(* PLC project testproj, Beckhoff Automation GmbH TwinCAT PLC Control 3.5.20.50 *)
(* stored: creationDateTime 2025-07-01T11:02:16.1300929, modificationDateTime 2025-07-01T11:02:16.1300929 *)

FUNCTION_BLOCK AnaMon
  VAR_INPUT
    WQC : BYTE;
    OSLevel : BYTE;
    V : REAL;
    VSclMin : REAL;
    VSclMax : REAL;
    VUnit : INT;
    VAHEn : BOOL;
    VWHEn : BOOL;
    VTHEn : BOOL;
    VTLEn : BOOL;
    VWLEn : BOOL;
    VALEn : BOOL;
  END_VAR
  VAR_OUTPUT
    VAHAct : BOOL;
    VWHAct : BOOL;
    VTHAct : BOOL;
    VTLAct : BOOL;
    VWLAct : BOOL;
    VALAct : BOOL;
  END_VAR
  VAR
    VAHLim : REAL;
    VWHLim : REAL;
    VTHLim : REAL;
    VTLLim : REAL;
    VWLLim : REAL;
    VALLim : REAL;
  END_VAR

            
// Copy MTP base variables to local temporaries (READ access)


VAHAct := vOut >= alarmHigh;
VWHAct := vOut >= warningHigh;
VTHAct := vOut >= toleranceHigh;
VTLAct := vOut <= toleranceLow;
VWLAct := vOut <= warningLow;
VALAct := vOut <= alarmLow;

// Copy local temporaries back to MTP base variables (WRITE access)

        
END_FUNCTION_BLOCK

FUNCTION_BLOCK BinMon
  VAR_INPUT
    wQC : BYTE;
    vState0 : STRING;
    vState1 : STRING;
    oSLevel : BYTE;
    vFlutEn : BOOL;
  END_VAR
  VAR_OUTPUT
    vFlutAct : BOOL;
  END_VAR
  VAR
    vFlutCnt : INT;
  END_VAR

            
// Copy MTP base variables to local temporaries (READ access)



// Copy local temporaries back to MTP base variables (WRITE access)

        
END_FUNCTION_BLOCK

FUNCTION_BLOCK LockView4
  VAR_INPUT
    wQC : BYTE;
    logic : BOOL;
    in1En : BOOL;
    in1 : BOOL;
    in1QC : BYTE;
    in1Inv : BOOL;
    in1Txt : STRING;
    in2En : BOOL;
    in2 : BOOL;
    in2QC : BYTE;
    in2Inv : BOOL;
    in2Txt : STRING;
    in3En : BOOL;
    in3 : BOOL;
    in3QC : BYTE;
    in3Inv : BOOL;
    in3Txt : STRING;
    in4En : BOOL;
    in4 : BOOL;
    in4QC : BYTE;
    in4Inv : BOOL;
    in4Txt : STRING;
  END_VAR
  VAR_OUTPUT
    out : BOOL;
    outQC : STRING;
  END_VAR

            
// Copy MTP base variables to local temporaries (READ access)



// Copy local temporaries back to MTP base variables (WRITE access)

        
END_FUNCTION_BLOCK

FUNCTION_BLOCK MonAnaDrv

            
// Copy MTP base variables to local temporaries (READ access)



// Copy local temporaries back to MTP base variables (WRITE access)

        
END_FUNCTION_BLOCK

FUNCTION_BLOCK MonAnaVlv

            
// Copy MTP base variables to local temporaries (READ access)



// Copy local temporaries back to MTP base variables (WRITE access)

        
END_FUNCTION_BLOCK

FUNCTION_BLOCK MonBinDrv
  VAR_INPUT
    stateChannel : BOOL;
    stateOffAut : BOOL;
    stateOpAut : BOOL;
    stateAutAut : BOOL;
    permit : BOOL;
    intlEn : BOOL;
    interlock : BOOL;
    protEn : BOOL;
    protect : BOOL;
    wQC : BYTE;
    oSLevel : BYTE;
    safePos : BOOL;
    fwdEn : BOOL;
    revEn : BOOL;
    stopAut : BOOL;
    fwdAut : BOOL;
    revAut : BOOL;
    revFbkCalc : BOOL;
    revFbk : BOOL;
    fwdFbkCalc : BOOL;
    fwdFbk : BOOL;
    trip : BOOL;
    resetAut : BOOL;
    monSafePos : BOOL;
    monStatTi : REAL;
    monDynTi : REAL;
  END_VAR
  VAR_OUTPUT
    stateOpAct : BOOL;
    stateAutAct : BOOL;
    stateOffAct : BOOL;
    safePosAct : BOOL;
    fwdCtrl : BOOL;
    revCtrl : BOOL;
    monStatErr : BOOL;
    monDynErr : BOOL;
  END_VAR
  VAR
    stateOffOp : BOOL;
    stateOpOp : BOOL;
    stateAutOp : BOOL;
    stopOp : BOOL;
    fwdOp : BOOL;
    revOp : BOOL;
    resetOp : BOOL;
    monEn : BOOL;
  END_VAR

            
// Copy MTP base variables to local temporaries (READ access)



// Copy local temporaries back to MTP base variables (WRITE access)

        
END_FUNCTION_BLOCK

FUNCTION_BLOCK MonBinVlv
  VAR_INPUT
    StateChannel : BOOL;
    StateOffAut : BOOL;
    StateOpAut : BOOL;
    StateAutAut : BOOL;
    PermEn : BOOL;
    IntlEn : BOOL;
    ProtEn : BOOL;
    Permit : BOOL;
    Interlock : BOOL;
    Protect : BOOL;
    WQC : BYTE;
    SafePos : BOOL;
    OpenAut : BOOL;
    CloseAut : BOOL;
    OpenFbkCalc : BOOL;
    CloseFbkCalc : BOOL;
    OpenFbk : BOOL;
    CloseFbk : BOOL;
    MonSafePos : BOOL;
    MonStatTi : REAL;
    MonDynTi : REAL;
    ResetAut : BOOL;
  END_VAR
  VAR_OUTPUT
    StateOpAct : BOOL;
    StateAutAct : BOOL;
    StateOffAct : BOOL;
    SafePosAct : BOOL;
    Ctrl : BOOL;
    MonStatErr : BOOL;
    MonDynErr : BOOL;
    OperationMode : INT;
  END_VAR
  VAR
    StateOffOp : BOOL;
    StateOpOp : BOOL;
    StateAutOp : BOOL;
    OpenOp : BOOL;
    CloseOp : BOOL;
    ResetOp : BOOL;
    MonEn : BOOL;
    OpenedState : BOOL;
    ClosedState : BOOL;
    DelayTimer1 : TON;
    DelayTimer2 : TON;
  END_VAR

            
// Copy MTP base variables to local temporaries (READ access)


    
// State Machine for the OperationMode
CASE OperationMode OF
    0: // Offline
        IF (StateOpAut AND StateChannel) OR (StateOpOp AND NOT StateChannel) THEN
            OperationMode := 1;
        END_IF;
    1: // Operator
        IF (StateOffAut AND StateChannel) OR (StateOffOp AND NOT StateChannel) THEN
            OperationMode := 0;
        END_IF;
        IF (StateAutAut AND StateChannel) OR (StateAutOp AND NOT StateChannel) THEN
            OperationMode := 2;
        END_IF;
    2: // Automatic
        IF (StateOpAut AND StateChannel) OR (StateOpOp AND NOT StateChannel) THEN
            OperationMode := 1;
        END_IF;
END_CASE;
    
// Make boolean indicators for the OperationMode State
StateOpAct := OperationMode = 1;
StateAutAct := OperationMode = 2;
StateOffAct := OperationMode = 0;
    
// 'Protect' is for interlocks that need to be reset
IF (ResetAut AND StateChannel) OR (ResetOp AND NOT StateChannel) THEN
    Protect := FALSE;
END_IF;
    
// signal indicating that the valve needs to go to the safe position
SafePosAct := (PermEn AND NOT Permit) OR (IntlEn AND NOT Interlock) OR (ProtEn AND NOT Protect) OR (MonEn AND (MonStatErr OR MonDynErr));
    
// control signal to the hardware
IF (SafePosAct AND SafePos AND NOT SafePosEn) OR (NOT SafePosAct AND ((OpenAut AND StateAutAct) OR (OpenOp and StateOpAct))) THEN
    Ctrl := TRUE;
END_IF;
IF (SafePosAct AND NOT SafePos NOT SafePosEn) OR (NOT SafePosAct AND ((CloseAut AND StateAutAct) OR (CloseOp and StateOpAct))) THEN
    Ctrl := FALSE;
END_IF;
    
// Opened and Closed States
IF Ctrl AND OpenFbk THEN
    OpenedState := TRUE;
END_IF;
IF NOT Ctrl THEN
    OpenedState := FALSE;
END_IF;
IF NOT Ctrl AND CloseFbk THEN
    ClosedState := TRUE;
END_IF;
IF Ctrl THEN
    ClosedState := FALSE;
END_IF;
    
// Static and Dynamic Monitoring
DelayTimer1(IN:= (MonEn AND OpenedState AND NOT OpenFbk) OR ( MonEn AND ClosedState AND NOT CloseFbk), PT:= REAL_TO_TIME(MonStatTi * 1000));
IF DelayTimer1.Q THEN
    MonStatErr := TRUE;
END_IF;
IF (ResetAut AND StateChannel) OR (ResetOp AND NOT StateChannel) THEN
    MonStatErr := FALSE;
END_IF;
DelayTimer2(IN:= MonEn AND ((Ctrl AND NOT OpenFbk) OR (NOT Ctrl AND NOT ClsFbk)), PT:= REAL_TO_TIME(MonDynTi * 1000));
IF DelayTimer2.Q THEN
    MonDynErr := TRUE;
END_IF;
IF (ResetAut AND StateChannel) OR (ResetOp AND NOT StateChannel) THEN
    MonDynErr := FALSE;
END_IF;
    
// reset operator command
StateOffOp := False;
StateOpOp := False;
StateAutOp := False;
OpenOp := False;
CloseOp := False;
ResetOp := False;
    

// Copy local temporaries back to MTP base variables (WRITE access)

        
END_FUNCTION_BLOCK

FUNCTION_BLOCK PIDCtrl

            
// Copy MTP base variables to local temporaries (READ access)



// Copy local temporaries back to MTP base variables (WRITE access)

        
END_FUNCTION_BLOCK

FUNCTION_BLOCK AnalogInput
  VAR_INPUT
    rawValue : WORD;
    valueUnit : INT;
    scaleMin : REAL;
    scaleMax : REAL;
    alarmHigh : REAL;
    warningHigh : REAL;
    toleranceHigh : REAL;
    toleranceLow : REAL;
    warningLow : REAL;
    alarmLow : REAL;
    alarmHighEn : BOOL;
    warningHighEn : BOOL;
    toleranceHighEn : BOOL;
    toleranceLowEn : BOOL;
    warningLowEn : BOOL;
    alarmLowEn : BOOL;
  END_VAR
  VAR_OUTPUT
    alarmHighAct : REAL;
    warningHighAct : REAL;
    toleranceHighAct : REAL;
    toleranceLowAct : REAL;
    warningLowAct : REAL;
    alarmLowAct : REAL;
  END_VAR

            
// Copy MTP base variables to local temporaries (READ access)


WQC := 16#FF;
OSLevel := TODO;
V := scaleMin + (REAL(RawInput) / 27648.0) * (scaleMax - scaleMin);
vOut := V;
VSclMin := scaleMin;
VSclMax := scaleMax;
VUnit := valueUnit;
alarmHigh := VAHLim;
warningHigh := VWHLim;
toleranceHigh := VTHLim;
toleranceLow := VTLLim;
warningLow := VWLLim;
alarmLow := VALLim;
VAHEn := alarmHighEn;
VWHEn := warningHighEn;
VTHEn := toleranceHighEn;
VTLEn := toleranceLowEn;
VWLEn := warningLowEn;
VALEn := alarmLowEn;
    
    

// Copy local temporaries back to MTP base variables (WRITE access)

        
END_FUNCTION_BLOCK

FUNCTION_BLOCK AnalogValve

            
// Copy MTP base variables to local temporaries (READ access)



// Copy local temporaries back to MTP base variables (WRITE access)

        
END_FUNCTION_BLOCK

FUNCTION_BLOCK DigitalInput

            
// Copy MTP base variables to local temporaries (READ access)



// Copy local temporaries back to MTP base variables (WRITE access)

        
END_FUNCTION_BLOCK

FUNCTION_BLOCK Interlock4

            
// Copy MTP base variables to local temporaries (READ access)



// Copy local temporaries back to MTP base variables (WRITE access)

        
END_FUNCTION_BLOCK

FUNCTION_BLOCK PIDController

            
// Copy MTP base variables to local temporaries (READ access)



// Copy local temporaries back to MTP base variables (WRITE access)

        
END_FUNCTION_BLOCK

FUNCTION_BLOCK ReversingMotor

            
// Copy MTP base variables to local temporaries (READ access)



// Copy local temporaries back to MTP base variables (WRITE access)

        
END_FUNCTION_BLOCK

FUNCTION_BLOCK SolenoidValve
  VAR_IN_OUT
    MTPBase : FB_MTP_MonBinVlv;
  END_VAR
  VAR_INPUT
    id : INT;
    open : BOOL;
    close : BOOL;
    feedbackOpen : BOOL;
    feedbackClose : BOOL;
    hasFbOpen : BOOL;
    hasFbClose : BOOL;
    safeOpen : BOOL;
    safeHold : BOOL;
    monitor : BOOL;
    simulate : BOOL;
    simulateDelay : BOOL;
    interlockIn : BOOL;
    permitIn : BOOL;
    protectIn : BOOL;
    reset : BOOL;
  END_VAR
  VAR_OUTPUT
    remote : BOOL;
    operator : BOOL;
    automatic : BOOL;
    offline : BOOL;
    error : BOOL;
    opened : BOOL;
    closed : BOOL;
  END_VAR
  VAR
    fbOpenSimulated : BOOL;
    fbCloseSimulated : BOOL;
    DelayTimer1 : TON;
    DelayTimer2 : TON;
    StateChannel : BOOL;
    StateOpAct : BOOL;
    StateAutAct : BOOL;
    StateOffAct : BOOL;
    PermEn : BOOL;
    IntlEn : BOOL;
    ProtEn : BOOL;
    Permit : BOOL;
    Interlock : BOOL;
    Protect : BOOL;
    WQC : BYTE;
    SafePos : BOOL;
    OpenAut : BOOL;
    CloseAut : BOOL;
    Ctrl : BOOL;
    OpenFbkCalc : BOOL;
    CloseFbkCalc : BOOL;
    OpenFbk : BOOL;
    CloseFbk : BOOL;
    MonSafePos : BOOL;
    ResetAut : BOOL;
    MonEn : BOOL;
  END_VAR

            
// Copy MTP base variables to local temporaries (READ access)
StateChannel := MTPBase.StateChannel;
StateOpAct := MTPBase.StateOpAct;
StateAutAct := MTPBase.StateAutAct;
StateOffAct := MTPBase.StateOffAct;
Ctrl := MTPBase.Ctrl;
OpenFbk := MTPBase.OpenFbk;
CloseFbk := MTPBase.CloseFbk;


WQC := 16#FF;
OSLevel := TODO;
remote := StateChannel;
operator := StateOpAct;
automatic := StateAutAct;
offline := StateOffAct;
PermEn := True;
IntlEn := True;
ProtEn := True;
Permit := permitIn;
Interlock := interlockIn;
IF protectIn THEN
    Protect := TRUE;
END_IF;
SafePos := safeOpen;
MonSafePos := safeOpen;
SafePosEn := safeHold;
OpenAut := open;
CloseAut := close;
OpenFbkCalc := simulation OR NOT feedbackOpen;
CloseFbkCalc := simulation OR NOT feedbackClose;
DelayTimer1(IN:= (simulate OR NOT hasFbOpen) AND Ctrl, PT:= REAL_TO_TIME(simulateDelay * 1000));
fbOpenSimulated := DelayTimer1.Q;
DelayTimer2(IN:= (simulate OR NOT hasFbClose) AND NOT Ctrl, PT:= REAL_TO_TIME(simulateDelay * 1000));
fbCloseSimulated := DelayTimer2.Q;
OpenFbk := feedbackOpen OR fbOpenSimulated;
CloseFbk := feedbackClose OR fbCloseSimulated;
opened := Ctrl AND OpenFbk;
closed := NOT Ctrl AND CloseFbk;
ResetAut := reset;
MonEn := monitor;
reset := False;

// Copy local temporaries back to MTP base variables (WRITE access)
MTPBase.PermEn := PermEn;
MTPBase.IntlEn := IntlEn;
MTPBase.ProtEn := ProtEn;
MTPBase.Permit := Permit;
MTPBase.Interlock := Interlock;
MTPBase.Protect := Protect;
MTPBase.WQC := WQC;
MTPBase.SafePos := SafePos;
MTPBase.OpenAut := OpenAut;
MTPBase.CloseAut := CloseAut;
MTPBase.OpenFbkCalc := OpenFbkCalc;
MTPBase.CloseFbkCalc := CloseFbkCalc;
MTPBase.OpenFbk := OpenFbk;
MTPBase.CloseFbk := CloseFbk;
MTPBase.MonSafePos := MonSafePos;
MTPBase.ResetAut := ResetAut;
MTPBase.MonEn := MonEn;

        
END_FUNCTION_BLOCK

FUNCTION_BLOCK VFD

            
// Copy MTP base variables to local temporaries (READ access)



// Copy local temporaries back to MTP base variables (WRITE access)

        
END_FUNCTION_BLOCK
